Fanuc TP program (LS listing): MOVE2PERCH90.LS

/PROG  MOVE2PERCH90
/ATTR
OWNER		= MNEDITOR;
COMMENT		= "macro perch 90";
PROG_SIZE	= 267;
CREATE		= DATE 19-10-01  TIME 17:54:46;
MODIFIED	= DATE 19-10-01  TIME 17:55:20;
FILE_NAME	= MOVE2PER;
VERSION		= 0;
LINE_COUNT	= 4;
MEMORY_SIZE	= 623;
PROTECT		= READ_WRITE;
TCD:  STACK_SIZE	= 0,
      TASK_PRIORITY	= 50,
      TIME_SLICE	= 0,
      BUSY_LAMP_OFF	= 0,
      ABORT_REQUEST	= 0,
      PAUSE_REQUEST	= 0;
DEFAULT_GROUP	= 1,*,*,*,*;
CONTROL_CODE	= 00000000 00000000;
/APPL
/APPL

AUTO_SINGULARITY_HEADER;
  ENABLE_SINGULARITY_AVOIDANCE   : TRUE;
/MN
   1:  !Set UT & UF ;
   2:  UTOOL_NUM=1 ;
   3:  UFRAME_NUM=1 ;
   4:J PR[16:Perch90] 100% FINE    ;
/POS
/END
